// A collection whose access/mutation of items is last-in, first-out.
{attribute 'enable_dynamic_creation'}
{attribute 'no_assign'}
{attribute 'no_explicit_call' := 'direct call for this function block is not allowed'}
FUNCTION_BLOCK FB_Stack IMPLEMENTS I_Stack //, I_Enumerable, I_Copyable
VAR
	fbList : FB_List;
END_VAR

// Number of items in the collection.
PROPERTY _Count : T_Capacity
GET
_Count := THIS^.fbList._Count;
END_GET
END_PROPERTY

// Checks if collection is empty.
PROPERTY _Empty : BOOL
GET
_Empty := THIS^.fbList._Empty;
END_GET
END_PROPERTY

// Error status of the collection.
PROPERTY _Error_Status : T_Error
GET
_Error_Status := THIS^.fbList._Error_Status;
END_GET
END_PROPERTY

// Gets an immutable list of the items in the stack.
PROPERTY _Values : I_Immutable_List
GET
VAR_INST
	fbImmutable_List : FB_Immutable_List := (ipList := THIS^.fbList);
END_VAR
_Values := fbImmutable_List;
END_GET
END_PROPERTY

// Empties/Clears/Deletes every item in the stack.
METHOD Clear : I_Stack
Clear := THIS^;

THIS^.fbList.Clear();
END_METHOD

// Gets item at the top of the stack.
METHOD Get : I_Stack
VAR_INPUT
	Item : ANY; // Variable to store returned item value. 
END_VAR
VAR_OUTPUT
	bSuccess : BOOL;
END_VAR
Get := THIS^;

THIS^.fbList.Get(0, Item, bSuccess => bSuccess);
END_METHOD

// Gets item at the top of the stack as a generic.
METHOD Get_Generic : I_Stack
VAR_OUTPUT
	Item : T_Generic; // Variable to store returned item value
	bSuccess : BOOL;
END_VAR
Get_Generic := THIS^;

THIS^.fbList.Get_Generic(0, Item => Item, bSuccess => bSuccess);
END_METHOD

// Removes item at the top of the stack without returning anything.
METHOD Pop : I_Stack
VAR_OUTPUT
	bSuccess : BOOL;
END_VAR
Pop := THIS^;

THIS^.fbList.Remove_At(0, bSuccess => bSuccess);
END_METHOD

// Add item to the top of the stack.
METHOD Push : I_Stack
VAR_INPUT
	Item : ANY; // Item to store.
END_VAR
VAR_OUTPUT
	bSuccess : BOOL;
END_VAR
Push := THIS^;

THIS^.fbList.Insert_Generic(0, Item, bSuccess => bSuccess);
END_METHOD

// Add generic item to the top of the stack.
METHOD Push_Generic : I_Stack
VAR_INPUT
	Item : T_Generic; // Item to store.
END_VAR
VAR_OUTPUT
	bSuccess : BOOL;
END_VAR
Push_Generic := THIS^;

THIS^.fbList.Insert_Generic(0, Item, bSuccess => bSuccess);
END_METHOD

// Reverses order of items on stack.
METHOD Reverse : I_Stack
VAR_OUTPUT
	bSuccess : BOOL;
END_VAR
Reverse := THIS^;

THIS^.fbList.Reverse(bSuccess => bSuccess);
END_METHOD

END_FUNCTION_BLOCK

(* stored: Version 1.1.0.1
   POU FB_Stack: Id {9a992fe7-0267-06d4-33ff-969f591448bf}, SpecialFunc None
   Property _Count: Id {e3da9272-2181-0fd7-31c6-e44f0ef9d940}
   Get Get: Id {e4d5dc7b-be9b-097f-0188-b766c46c9a27}
   Property _Empty: Id {f47be231-0e01-054e-0e62-17967f9c9812}
   Get Get: Id {8d493fe3-cb73-0eef-3ff1-5b181590dff0}
   Property _Error_Status: Id {ed3158fd-9c54-086f-0317-fe3281e9a94e}
   Get Get: Id {6b3c95b7-43db-0123-0333-80ed36e54c60}
   Property _Values: Id {ac73bae5-8dcb-0d37-36e6-ab46adea9629}
   Get Get: Id {80ba323c-77b8-08bf-0dda-571a924acf61}
   Method Clear: Id {0eb2a151-1239-08ae-07d3-3463619cbdd7}
   Method Get: Id {3c7972ee-62a2-061d-1590-3cbee4ff11d5}
   Method Get_Generic: Id {8d0f459f-0065-01c0-2a59-65e8f17e91e4}
   Method Pop: Id {5b334a56-0cb9-09e3-1d10-c6f0aa505e90}
   Method Push: Id {2c6bbbe5-a3d2-00b6-15e3-2cd0292b435f}
   Method Push_Generic: Id {9150115e-0116-02eb-28f6-b7be4becb93e}
   Method Reverse: Id {84b66e32-e6a1-031d-03aa-5aa15541e96d} *)
